(* IEC 61131-3 sources: SRCI/RobotLibrary/RobotLibrary/POUs/General/MC_RobotTask (part 2) *)

      IF (Telegram.RobToPlc.Sequence[0].Fragment[0].Header.PayloadLength > 0)
      THEN
        // Fill Respone payload
        FOR _idx := Telegram.RobToPlc.Sequence[0].Fragment[0].Header.PayloadPointer TO Telegram.RobToPlc.Sequence[0].Fragment[0].Header.PayloadLength
        DO
          Telegram.RobToPlc.Sequence[0].Fragment[0].Command.Payload[_idx] := RecvData.GetByte();
        END_FOR

        // Add Response to ACR
        AxesGroup.Acyclic.ActiveCommandRegister.AddRsp(Telegram.RobToPlc.Sequence[0].Fragment[0]);

        // Only for debugging
        Telegram.RobToPlc.Sequence[0].Fragment[0].Command.Header.State                 := GetHalfeByteLo(Telegram.RobToPlc.Sequence[0].Fragment[0].Command.Payload[0]);
        Telegram.RobToPlc.Sequence[0].Fragment[0].Command.Header.ParSeq                := GetHalfeByteHi(Telegram.RobToPlc.Sequence[0].Fragment[0].Command.Payload[0]);
        Telegram.RobToPlc.Sequence[0].Fragment[0].Command.Header.AlarmMessageSeverity  :=  BYTE_TO_SINT(Telegram.RobToPlc.Sequence[0].Fragment[0].Command.Payload[1]);
        Telegram.RobToPlc.Sequence[0].Fragment[0].Command.Header.AlarmMessageCode      :=  CombineBytesToUint( HiByte := Telegram.RobToPlc.Sequence[0].Fragment[0].Command.Payload[2],
                                                                                                               LoByte := Telegram.RobToPlc.Sequence[0].Fragment[0].Command.Payload[3]);
        // Create log entry
        CreateLogMessagePara5 ( Timestamp   := SystemTime,
                                MessageType := MessageType.CMD,
                                Severity    := Severity.DEBUG,
                                MessageCode := 0,
                                MessageText := 'RecvData: received Fragment [{1}] with PayloadLength = {2}, CmdID <{3}> , CmdState: {4}, Fragment-Action Bits: {5}',
                                Para1       :=  DINT_TO_STRING(0), {warning 'Add seqIdx'}
                                Para2       :=  UINT_TO_STRING            (Telegram.RobToPlc.Sequence[0].Fragment[0].Header.PayloadLength),
                                Para3       :=  DINT_TO_STRING            (Telegram.RobToPlc.Sequence[0].Fragment[0].Header.CmdID),
                                Para4       :=  CmdMessageStateToString   (Telegram.RobToPlc.Sequence[0].Fragment[0].Command.Header.State),
                                Para5       :=  ByteToFragmentActionString(Telegram.RobToPlc.Sequence[0].Fragment[0].Header.FragmentAction));
                                //Para6       :=  BYTE_TO_STRING(Telegram.RobToPlc.Header.LifeSign)
      END_IF
    END_IF
  END_IF

  {warning 'ToDo'}
  Telegram.RobToPlc.Footer.Reserve_LifeSign.0 := RecvData.Payload[255].4;
  Telegram.RobToPlc.Footer.Reserve_LifeSign.1 := RecvData.Payload[255].5;
  Telegram.RobToPlc.Footer.Reserve_LifeSign.2 := RecvData.Payload[255].6;
  Telegram.RobToPlc.Footer.Reserve_LifeSign.3 := RecvData.Payload[255].7;

  IF ( RobotLibraryParameter.TWO_SEQUENCES )
  THEN
   _seqCount := _seqCount + 1;
  END_IF

  AxesGroup.InternalData.LastACK[0] := Telegram.RobToPlc.Sequence[0].Header.SEQ_ACK; {warning 'ToDo Handle 2nd sequence'}

END_METHOD

METHOD PRIVATE ParseRecvPayloadCyclic
VAR_IN_OUT
  /// Robot assignment of function
  AxesGroup: AxesGroup;
END_VAR

END_METHOD

METHOD PRIVATE ParseRecvPayloadCyclicOptional
VAR_IN_OUT
  /// Robot assignment of function
  AxesGroup    : AxesGroup;
END_VAR

VAR
  /// internal index for loops
 _idx : DINT;
END_VAR

  // AxesGroup.OptionalCyclic.RobToPlc.SubProgramData {{{
  IF ( AxesGroup.CyclicOptional.RobToPlc.SubProgramData.Active )
  THEN
    FOR _idx := 0 TO 25 {warning 'Add contant for DataMax'}
    DO
      Telegram.RobToPlc.CyclicOptional.SubProgramData.Data[_idx] := RecvData.GetByte();
  	END_FOR
  END_IF
  // }}}

  // AxesGroup.OptionalCyclic.RobToPlc.CartesianPos {{{
  IF ( AxesGroup.CyclicOptional.RobToPlc.CartesianPosition.Active )
  THEN
    Telegram.RobToPlc.CyclicOptional.CartesianPosition.X                    := RecvData.GetReal();
    Telegram.RobToPlc.CyclicOptional.CartesianPosition.Y                    := RecvData.GetReal();
    Telegram.RobToPlc.CyclicOptional.CartesianPosition.Z                    := RecvData.GetReal();
    Telegram.RobToPlc.CyclicOptional.CartesianPosition.Rx                   := RecvData.GetReal();
    Telegram.RobToPlc.CyclicOptional.CartesianPosition.Ry                   := RecvData.GetReal();
    Telegram.RobToPlc.CyclicOptional.CartesianPosition.Rz                   := RecvData.GetReal();
    Telegram.RobToPlc.CyclicOptional.CartesianPosition.Config               := RecvData.GetWord();
    Telegram.RobToPlc.CyclicOptional.CartesianPosition.Turns_J2_J1          := RecvData.GetByte();
    Telegram.RobToPlc.CyclicOptional.CartesianPosition.Turns_J4_J3          := RecvData.GetByte();
    Telegram.RobToPlc.CyclicOptional.CartesianPosition.Turns_J6_J5          := RecvData.GetByte();
    Telegram.RobToPlc.CyclicOptional.CartesianPosition.Turns_E1             := RecvData.GetByte();
    Telegram.RobToPlc.CyclicOptional.CartesianPosition.E1                   := RecvData.GetReal();
    Telegram.RobToPlc.CyclicOptional.CartesianPosition.ToolNo               := RecvData.GetUsint();
    Telegram.RobToPlc.CyclicOptional.CartesianPosition.FrameNo              := RecvData.GetUsint();
    Telegram.RobToPlc.CyclicOptional.CartesianPosition.CurrentlyUsedToolNo  := RecvData.GetUsint();
    Telegram.RobToPlc.CyclicOptional.CartesianPosition.CurrentlyUsedFrameNo := RecvData.GetUsint();
    Telegram.RobToPlc.CyclicOptional.CartesianPosition.Reserve_1            := RecvData.GetByte();
    Telegram.RobToPlc.CyclicOptional.CartesianPosition.Reserve_2            := RecvData.GetByte();
  END_IF
  // }}}

  // AxesGroup.OptionalCyclic.RobToPlc.JointPosition {{{
  IF ( AxesGroup.CyclicOptional.RobToPlc.JointPosition.Active )
  THEN
    Telegram.RobToPlc.CyclicOptional.JointPosition.J1         := RecvData.GetReal();
    Telegram.RobToPlc.CyclicOptional.JointPosition.J2         := RecvData.GetReal();
    Telegram.RobToPlc.CyclicOptional.JointPosition.J3         := RecvData.GetReal();
    Telegram.RobToPlc.CyclicOptional.JointPosition.J4         := RecvData.GetReal();
    Telegram.RobToPlc.CyclicOptional.JointPosition.J5         := RecvData.GetReal();
    Telegram.RobToPlc.CyclicOptional.JointPosition.J6         := RecvData.GetReal();
    Telegram.RobToPlc.CyclicOptional.JointPosition.E1         := RecvData.GetReal();
    Telegram.RobToPlc.CyclicOptional.JointPosition.E1_Reserve := RecvData.GetWord();
  END_IF
  // }}}

  // AxesGroup.OptionalCyclic.RobToPlc.CartesianForce {{{
  IF ( AxesGroup.CyclicOptional.RobToPlc.Force.Active )
  THEN
    Telegram.RobToPlc.CyclicOptional.Force.X  := RecvData.GetReal();
    Telegram.RobToPlc.CyclicOptional.Force.Y  := RecvData.GetReal();
    Telegram.RobToPlc.CyclicOptional.Force.Z  := RecvData.GetReal();
    Telegram.RobToPlc.CyclicOptional.Force.Rx := RecvData.GetReal();
    Telegram.RobToPlc.CyclicOptional.Force.Ry := RecvData.GetReal();
    Telegram.RobToPlc.CyclicOptional.Force.Rz := RecvData.GetReal();
  END_IF
  // }}}

  // AxesGroup.OptionalCyclic.RobToPlc.Current {{{
  IF ( AxesGroup.CyclicOptional.RobToPlc.Current.Active )
  THEN
    Telegram.RobToPlc.CyclicOptional.Current.J1  := RecvData.GetReal();
    Telegram.RobToPlc.CyclicOptional.Current.J2  := RecvData.GetReal();
    Telegram.RobToPlc.CyclicOptional.Current.J3  := RecvData.GetReal();
    Telegram.RobToPlc.CyclicOptional.Current.J4  := RecvData.GetReal();
    Telegram.RobToPlc.CyclicOptional.Current.J5  := RecvData.GetReal();
    Telegram.RobToPlc.CyclicOptional.Current.J6  := RecvData.GetReal();
  END_IF

  // AxesGroup.OptionalCyclic.RobToPlc.CartesianPosExt {{{
  IF ( AxesGroup.CyclicOptional.RobToPlc.CartesianPositionExt.Active )
  THEN
    Telegram.RobToPlc.CyclicOptional.CartesianPositionExt.E2 := RecvData.GetReal();
    Telegram.RobToPlc.CyclicOptional.CartesianPositionExt.E3 := RecvData.GetReal();
    Telegram.RobToPlc.CyclicOptional.CartesianPositionExt.E4 := RecvData.GetReal();
    Telegram.RobToPlc.CyclicOptional.CartesianPositionExt.E5 := RecvData.GetReal();
    Telegram.RobToPlc.CyclicOptional.CartesianPositionExt.E6 := RecvData.GetReal();
  END_IF
  // }}}

  // AxesGroup.OptionalCyclic.RobToPlc.JointPosition {{{
  IF ( AxesGroup.CyclicOptional.RobToPlc.JointPositionExt.Active )
  THEN
    Telegram.RobToPlc.CyclicOptional.JointPositionExt.E2 := RecvData.GetReal();
    Telegram.RobToPlc.CyclicOptional.JointPositionExt.E3 := RecvData.GetReal();
    Telegram.RobToPlc.CyclicOptional.JointPositionExt.E4 := RecvData.GetReal();
    Telegram.RobToPlc.CyclicOptional.JointPositionExt.E5 := RecvData.GetReal();
    Telegram.RobToPlc.CyclicOptional.JointPositionExt.E6 := RecvData.GetReal();
  END_IF
  // }}}

  // AxesGroup.OptionalCyclic.RobToPlc.CartesianForceExt {{{
  IF ( AxesGroup.CyclicOptional.RobToPlc.ForceExt.Active )
  THEN
    Telegram.RobToPlc.CyclicOptional.ForceExt.E1  := RecvData.GetReal();
    Telegram.RobToPlc.CyclicOptional.ForceExt.E2  := RecvData.GetReal();
    Telegram.RobToPlc.CyclicOptional.ForceExt.E3  := RecvData.GetReal();
    Telegram.RobToPlc.CyclicOptional.ForceExt.E4  := RecvData.GetReal();
    Telegram.RobToPlc.CyclicOptional.ForceExt.E5  := RecvData.GetReal();
    Telegram.RobToPlc.CyclicOptional.ForceExt.E6  := RecvData.GetReal();
  END_IF
  // }}}

  // AxesGroup.OptionalCyclic.RobToPlc.CurrentExt {{{
  IF ( AxesGroup.CyclicOptional.RobToPlc.CurrentExt.Active )
  THEN
    Telegram.RobToPlc.CyclicOptional.CurrentExt.E1  := RecvData.GetReal();
    Telegram.RobToPlc.CyclicOptional.CurrentExt.E2  := RecvData.GetReal();
    Telegram.RobToPlc.CyclicOptional.CurrentExt.E3  := RecvData.GetReal();
    Telegram.RobToPlc.CyclicOptional.CurrentExt.E4  := RecvData.GetReal();
    Telegram.RobToPlc.CyclicOptional.CurrentExt.E5  := RecvData.GetReal();
    Telegram.RobToPlc.CyclicOptional.CurrentExt.E6  := RecvData.GetReal();
  END_IF
  // }}}

END_METHOD

METHOD PRIVATE ParseRecvPayloadFooter
VAR_IN_OUT
  /// Robot assignment of function
  AxesGroup : AxesGroup;
END_VAR

  {warning 'ToDo: use index from ParCfg'}
  Telegram.RobToPlc.Footer.Reserve_LifeSign.0 := RecvData.Payload[255].4;
  Telegram.RobToPlc.Footer.Reserve_LifeSign.1 := RecvData.Payload[255].5;
  Telegram.RobToPlc.Footer.Reserve_LifeSign.2 := RecvData.Payload[255].6;
  Telegram.RobToPlc.Footer.Reserve_LifeSign.3 := RecvData.Payload[255].7;

END_METHOD

METHOD PRIVATE ParseRecvPayloadHeader
VAR_IN_OUT
  /// Robot assignment of function
  AxesGroup    : AxesGroup;
END_VAR

  // Version
  Telegram.RobToPlc.Header.SRCIVersion := ByteToVersion(RecvData.GetByte());
  // Connection alive signal
  Telegram.RobToPlc.Header.LifeSign    := RecvData.GetHalfeByte2(IncPayloadPtr := TRUE);
  // Reserved byte
  Telegram.RobToPlc.Header.Reserved       := RecvData.GetByte();
  // Initialization and Telegram control state
  Telegram.RobToPlc.Header.TelegramState  := RecvData.GetUsint();
  // Combination of various RA related states.
  Telegram.RobToPlc.Header.StatusRobotArm := RecvData.GetDword();
  // Actual override in percentage encoding
  Telegram.RobToPlc.Header.Override       := RecvData.GetUint();

END_METHOD

METHOD PRIVATE ParseRecvPayloadLogging
VAR_IN_OUT
  /// Robot assignment of function
  AxesGroup    : AxesGroup;
END_VAR

VAR
  /// internal sequence index for loops
  _seqIdx : DINT;
  /// internal fragment index for loops
  _fragIdx : DINT;
END_VAR

  RETURN;
  FOR _seqIdx := 0 TO AxesGroup.InternalData.SequenceCountRecv
  DO
    // check new data to receive ?
    IF ( Telegram.RobToPlc.Sequence[_seqIdx].Header.SEQ_ACK <> AxesGroup.InternalData.LastACK[_seqIdx])
    THEN
      // Check sequence payload > 0 ?
      IF (Telegram.RobToPlc.Sequence[_seqIdx].Header.PayloadLength > 0)
      THEN
        // Create log entry
        CreateLogMessagePara4 ( Timestamp   := SystemTime,
                                MessageType := MessageType.CMD,
                                Severity    := Severity.DEBUG,
                                MessageCode := 0,
                                MessageText := 'RecvData: ACK = {1}, received Sequence [{2}] with PayloadLength = {3}, Lifesign = {4}',
                                Para1       :=  UINT_TO_STRING(Telegram.RobToPlc.Sequence[_seqIdx].Header.SEQ_ACK),
                                Para2       :=  DINT_TO_STRING(_seqIdx),
                                Para3       :=  UINT_TO_STRING(Telegram.RobToPlc.Sequence[_seqIdx].Header.PayloadLength),
                                Para4       :=  BYTE_TO_STRING(Telegram.RobToPlc.Header.LifeSign));

        FOR _fragIdx := 0 TO AxesGroup.InternalData.FragmentCountRecv
        DO
          // Check fragment payload > 0 ?
          IF (Telegram.RobToPlc.Sequence[_seqIdx].Fragment[_fragIdx].Header.PayloadLength > 0)
          THEN
            // Create log entry
            CreateLogMessagePara5 ( Timestamp   := SystemTime,
                                    MessageType := MessageType.CMD,
                                    Severity    := Severity.DEBUG,
                                    MessageCode := 0,
                                    MessageText := 'RecvData: received Fragment [{1}] with PayloadLength = {2}, CmdID <{3}> , CmdState: {4}, Fragment-Action Bits: {5}',
                                    Para1       :=  DINT_TO_STRING(0), {warning 'Add seqIdx'}
                                    Para2       :=  UINT_TO_STRING            (Telegram.RobToPlc.Sequence[_seqIdx].Fragment[_fragIdx].Header.PayloadLength),
                                    Para3       :=  DINT_TO_STRING            (Telegram.RobToPlc.Sequence[_seqIdx].Fragment[_fragIdx].Header.CmdID),
                                    Para4       :=  CmdMessageStateToString   (Telegram.RobToPlc.Sequence[_seqIdx].Fragment[_fragIdx].Command.Header.State),
                                    Para5       :=  ByteToFragmentActionString(Telegram.RobToPlc.Sequence[_seqIdx].Fragment[_fragIdx].Header.FragmentAction));
          END_IF
        END_FOR
      END_IF
    END_IF
  END_FOR

END_METHOD

METHOD PRIVATE ParseRecvPayloadSequence
VAR_IN_OUT
  /// Robot assignment of function
  AxesGroup    : AxesGroup;
END_VAR

VAR
  /// internal index
 _idx             : DINT;
  /// temporary DWORD
 _tmpDword        : DWORD;
  /// length of data block
 _dataBlockLength : UINT;
  /// internal payload length
 _payLoadLen      : DWORD;
  /// internal payload pointer
 _payLoadPtr      : DWORD;
  /// sequence counter
 _seqCount        : DINT;
END_VAR

VAR_INST
  /// last received acknowledge
 _lastACK : ARRAY[0..1] OF UDINT;
END_VAR

  // Sequence Data
  Telegram.RobToPlc.Sequence[0].Header.SEQ_ACK       := RecvData.GetUint();
  Telegram.RobToPlc.Sequence[0].Header.PayloadLength := RecvData.GetUint();

  // check new data ?
  IF ( Telegram.RobToPlc.Sequence[0].Header.SEQ_ACK <> AxesGroup.InternalData.LastACK[0]) {warning 'ToDo Handle 2nd sequence'}
  THEN

    IF (Telegram.RobToPlc.Sequence[0].Header.PayloadLength > 0)
    THEN
      // Create log entry
      CreateLogMessagePara4 ( Timestamp   := SystemTime,
                              MessageType := MessageType.CMD,
                              Severity    := Severity.DEBUG,
                              MessageCode := 0,
                              MessageText := 'RecvData: ACK = {1}, received Sequence [{2}] with PayloadLength = {3}, Lifesign = {4}',
                              Para1       :=  UINT_TO_STRING(Telegram.RobToPlc.Sequence[0].Header.SEQ_ACK),
                              Para2       :=  DINT_TO_STRING(0), {warning 'Add seqIdx'}
                              Para3       :=  UINT_TO_STRING(Telegram.RobToPlc.Sequence[0].Header.PayloadLength),
                              Para4       :=  BYTE_TO_STRING(Telegram.RobToPlc.Header.LifeSign));

      Telegram.RobToPlc.Sequence[0].Fragment[0].Header.CmdID               := RecvData.GetUint();
      Telegram.RobToPlc.Sequence[0].Fragment[0].Header.Reserve             := RecvData.GetByte();
      Telegram.RobToPlc.Sequence[0].Fragment[0].Header.FragmentAction      := RecvData.GetByte();
      Telegram.RobToPlc.Sequence[0].Fragment[0].Header.PayloadPointer      := RecvData.GetUint();
      Telegram.RobToPlc.Sequence[0].Fragment[0].Header.PayloadLength       := RecvData.GetUint();

      IF (Telegram.RobToPlc.Sequence[0].Fragment[0].Header.PayloadLength > 0)
      THEN
        // Fill Respone payload
        FOR _idx := Telegram.RobToPlc.Sequence[0].Fragment[0].Header.PayloadPointer TO Telegram.RobToPlc.Sequence[0].Fragment[0].Header.PayloadLength
        DO
          Telegram.RobToPlc.Sequence[0].Fragment[0].Command.Payload[_idx] := RecvData.GetByte();
        END_FOR

        // Add Response to ACR
        AxesGroup.Acyclic.ActiveCommandRegister.AddRsp(Telegram.RobToPlc.Sequence[0].Fragment[0]);

        // Only for debugging
        Telegram.RobToPlc.Sequence[0].Fragment[0].Command.Header.State                 := GetHalfeByteLo(Telegram.RobToPlc.Sequence[0].Fragment[0].Command.Payload[0]);
        Telegram.RobToPlc.Sequence[0].Fragment[0].Command.Header.ParSeq                := GetHalfeByteHi(Telegram.RobToPlc.Sequence[0].Fragment[0].Command.Payload[0]);
        Telegram.RobToPlc.Sequence[0].Fragment[0].Command.Header.AlarmMessageSeverity  :=  BYTE_TO_SINT(Telegram.RobToPlc.Sequence[0].Fragment[0].Command.Payload[1]);
        Telegram.RobToPlc.Sequence[0].Fragment[0].Command.Header.AlarmMessageCode      :=  CombineBytesToUint( HiByte := Telegram.RobToPlc.Sequence[0].Fragment[0].Command.Payload[2],
                                                                                                               LoByte := Telegram.RobToPlc.Sequence[0].Fragment[0].Command.Payload[3]);
        // Create log entry
        CreateLogMessagePara5 ( Timestamp   := SystemTime,
                                MessageType := MessageType.CMD,
                                Severity    := Severity.DEBUG,
                                MessageCode := 0,
                                MessageText := 'RecvData: received Fragment [{1}] with PayloadLength = {2}, CmdID <{3}> , CmdState: {4}, Fragment-Action Bits: {5}',
                                Para1       :=  DINT_TO_STRING(0), {warning 'Add seqIdx'}
                                Para2       :=  UINT_TO_STRING            (Telegram.RobToPlc.Sequence[0].Fragment[0].Header.PayloadLength),
                                Para3       :=  DINT_TO_STRING            (Telegram.RobToPlc.Sequence[0].Fragment[0].Header.CmdID),
                                Para4       :=  CmdMessageStateToString   (Telegram.RobToPlc.Sequence[0].Fragment[0].Command.Header.State),
                                Para5       :=  ByteToFragmentActionString(Telegram.RobToPlc.Sequence[0].Fragment[0].Header.FragmentAction));
                                //Para6       :=  BYTE_TO_STRING(Telegram.RobToPlc.Header.LifeSign)
      END_IF
    END_IF
  END_IF

  IF ( RobotLibraryParameter.TWO_SEQUENCES ) {warning 'ToDo'}
  THEN
   _seqCount := _seqCount + 1;
  END_IF

END_METHOD
